FUNCTION CompAsITag : Result
VAR_INPUT
	iSource	: I_Component;
END_VAR
VAR_OUTPUT
	iDest	: I_Tag;
END_VAR

IF iSource = 0 THEN
	CompAsITag := Err.Itf0;
	RETURN;
END_IF

IF __QUERYINTERFACE(iSource, iDest) THEN
	CompAsITag := Ok;
ELSE
	CompAsITag := Err.NoMatch;
END_IF

END_FUNCTION

(* stored: Version 1.1.0.1
   POU CompAsITag: Id {3feb1b07-c695-429c-b10c-285305651b80}, SpecialFunc None *)
